TYPE ST_CAT :
STRUCT
	bValue0, 
	bValue1 : BOOL;
	fValue 	: REAL; 
END_STRUCT
END_TYPE

(* stored: Version 1.1.0.1, ProductVersion 3.1.4024.4
   DUT ST_CAT: Id {0762c699-fd93-4bc7-a1ae-cab90e2ddac8} *)
